Universal Robots PolyScope program: T01_remove_cover.urp

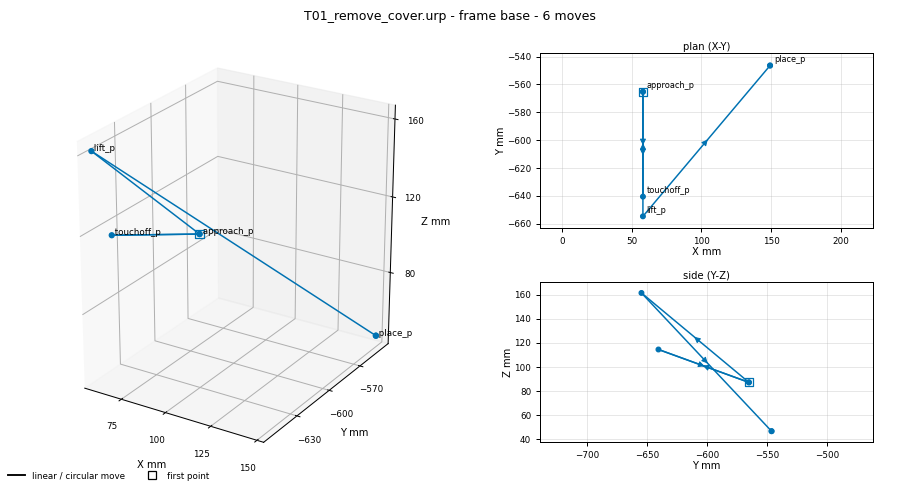
[picture p0: tool path of T01_remove_cover.urp in frame base, 6 of 7 moves have a stored position in this frame; points joined in program order, loops and branches not executed]
Program T01_remove_cover (installation=default directory=/programs createdIn=5.9.1.1031110 lastSavedIn=5.9.1.1031110 robotSerialNumber=20195501059)
Calibrated DH parameters: a=[0.000146, -0.418764, -0.053981, 0.000058, -0.000023, 0]; d=[0.162545, 37.319448, -206.067439, 168.881546, 0.09955, 0.099464]; alpha=[1.57004, -0.001979, 0.002304, 1.570607, -1.57066, 0]; deltaTheta=[0, -0.174616, -1.258233, 1.432844, -0.000001, 0]
BeforeStart
  URCap Gripper Activate (Robotiq_Grippers, Robotiq Inc.) dataModel(ResetAndActivateKey=false)
  start_p := get_actual_tcp_pose()
  MoveJ speed 60 deg/s, acceleration 80 deg/s^2 (useActiveTCP=true) feature=Base
    Waypoint Waypoint (Variable): variable=start_p
Robot Program (runOnlyOnce=true)
  MoveL speed 250 mm/s, acceleration 1200 mm/s^2 (useActiveTCP=true) feature=Base
    Waypoint approach_p: TCP in base x=58.113 y=-565.269 z=87.223 mm, rx=2.2518 ry=2.1907 rz=0.0001 rad; joints [82.25, -73.485, 105.724, -122.228, 270.032, 83.85] deg; TCP offset x=0 y=0 z=174 mm, rx=0 ry=0 rz=0 rad
    URCap Gripper (Robotiq_Grippers, Robotiq Inc.) dataModel(position=100.0, force=100.0, speed=100.0, positionInDouble=100.0, forceInDouble=100.0, speedInDouble=100.0, slaveIds=[9], blocking=false)
    Waypoint touchoff_p: TCP in base x=58.124 y=-640.467 z=114.561 mm, rx=2.2517 ry=2.1906 rz=0 rad; joints [83.174, -66.062, 90.614, -114.549, 270.005, 84.76] deg
    MoveDirectionNode (selectedDirection=ZPlus toolParams=0.01, 1.2) feature=Joint_6_name
      Until TOOL_CONTACT_DETECTION (allowActions=false retraction=0.002 decelerationAcceleration=3 decelerationAngularAcceleration=34.906585)
      Until DISTANCE (allowActions=true deceleration=3 distanceNodeType=STOP) Distance=0.01; motionParameters(blendRadius=0)
        MoveL speed 250 mm/s, acceleration 1200 mm/s^2 (useActiveTCP=true) feature=Base
          Waypoint approach_p: TCP in base x=58.113 y=-565.269 z=87.223 mm, rx=2.2518 ry=2.1907 rz=0.0001 rad; joints [82.25, -73.485, 105.724, -122.228, 270.032, 83.85] deg
        Halt
  URCap Gripper (Robotiq_Grippers, Robotiq Inc.) dataModel(position=55.0, force=100.0, speed=100.0, positionInDouble=55.0, forceInDouble=100.0, speedInDouble=100.0, slaveIds=[9], blocking=true)
  URCap Olis Teleop (Olis Teleop, Olis Robotics) dataModel(OperatorMessage=Please remove cover)
  MoveL speed 250 mm/s, acceleration 1200 mm/s^2 (useActiveTCP=true) feature=Base
    Waypoint lift_p: TCP in base x=58.101 y=-654.603 z=161.57 mm, rx=2.2517 ry=2.1905 rz=-0.0002 rad; joints [83.325, -66.526, 83.949, -107.429, 269.992, 84.904] deg
  MoveL speed 250 mm/s, acceleration 1200 mm/s^2 (useActiveTCP=true) feature=Base
    Waypoint place_p: TCP in base x=149.28 y=-546.453 z=46.637 mm, rx=2.2516 ry=2.1906 rz=-0.0002 rad; joints [91.614, -70.399, 108.627, -128.235, 270.035, 93.22] deg
    MoveDirectionNode (selectedDirection=ZPlus toolParams=0.02, 1.2) feature=Joint_6_name
      Until TOOL_CONTACT_DETECTION (allowActions=true retraction=0 decelerationAcceleration=3 decelerationAngularAcceleration=34.906585)
        URCap Gripper (Robotiq_Grippers, Robotiq Inc.) dataModel(position=55.0, force=100.0, speed=100.0, positionInDouble=55.0, forceInDouble=100.0, speedInDouble=100.0, slaveIds=[9], blocking=true)
        MoveDirectionNode (selectedDirection=ZPlus toolParams=0.02, 1.2) feature=Joint_6_name
          Until DISTANCE (allowActions=false deceleration=3 distanceNodeType=STOP) Distance=0.005; motionParameters(blendRadius=0)
      Until DISTANCE (allowActions=false deceleration=3 distanceNodeType=STOP) Distance=0.03; motionParameters(blendRadius=0)
    Waypoint place_p: motionParameters(blendRadius=0.05); TCP in base x=149.28 y=-546.453 z=46.637 mm, rx=2.2516 ry=2.1906 rz=-0.0002 rad; joints [91.614, -70.399, 108.627, -128.235, 270.035, 93.22] deg
    MoveDirectionNode (selectedDirection=ZMinus) feature=Joint_6_name
      Until DISTANCE (allowActions=false deceleration=3 distanceNodeType=STOP) Distance=0.025; motionParameters(blendRadius=0)
